INTERFACE ITmsMover EXTENDS IMover

METHOD ActivateTrack : BOOL
VAR_INPUT
	newTrack : OTCID;
END_VAR
END_METHOD

PROPERTY ActiveTrack : OTCID
GET
END_GET
END_PROPERTY

METHOD SetMoverInterface : BOOL
VAR_INPUT
	MoverInterface : I_TcIoXtsXpuMover;
END_VAR
END_METHOD

END_INTERFACE

(* stored: Version 1.1.0.1, ProductVersion 3.1.4024.12
   Itf ITmsMover: Id {1ee96f90-56ef-4744-a7ca-e48dd6e1711f}
   Method ActivateTrack: Id {d6312dcf-7ad6-4608-bca7-de68a24d417d}
   Property ActiveTrack: Id {f34bb9dc-3dd9-450b-b812-3982c42db988}
   Get Get: Id {398e1027-07bf-4a89-b2a9-b111367e8bbf}
   Method SetMoverInterface: Id {b8f5aad1-7a34-4096-9ecf-6a7b0f9a9c04} *)
